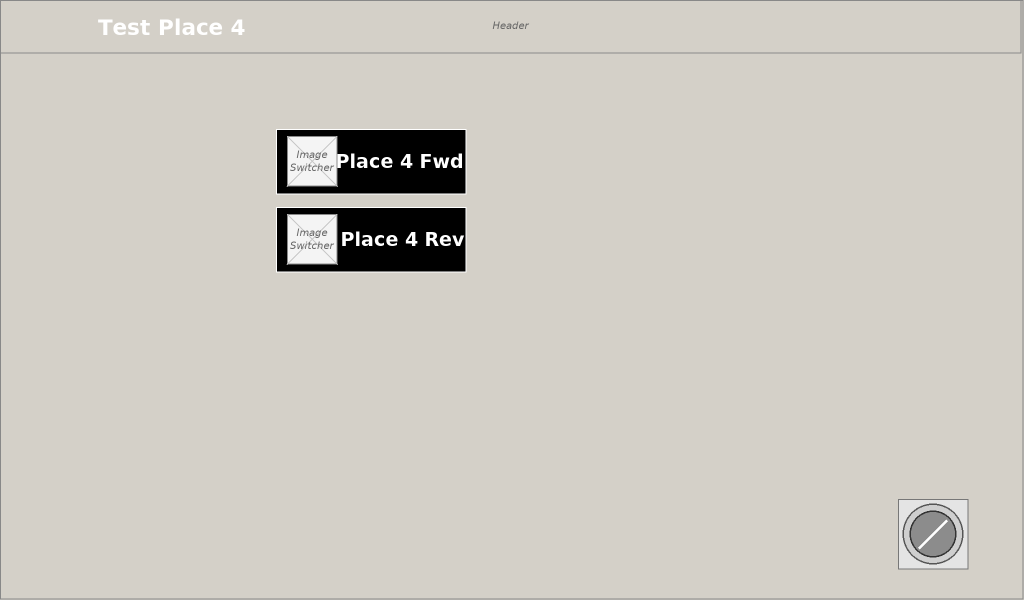
VISUALIZATION Test_Place4  // 1024x600
    Frame (0,-2 1021x55)
        shows Header()
    Label (95,15 250x25), "Test Place 4"
    RotarySwitch (898,499 70x70), variable: HMI_GVL.bTestModeEnablePlacing4, behaviour: TOGGLE, style: Switch-RotarySwitch-Gray
    RoundedRectangle (276,129 190x65)
        toggle Status_GVL.stMotor_Placing4.iTestForward
    Label (331,149 137x25), "Place 4 Fwd"
    ImageSwitcher (287,136 50x50), variable: Status_GVL.stMotor_Placing4.iTestForward, behaviour: TOGGLE
    RoundedRectangle (276,207 190x65)
        toggle Status_GVL.stMotor_Placing4.iTestReverse
    Label (334,227 137x25), "Place 4 Rev"
    ImageSwitcher (287,214 50x50), variable: Status_GVL.stMotor_Placing4.iTestReverse, behaviour: TOGGLE
END_VISUALIZATION

(* stored: Version 1.1.0.1, ProductVersion 3.1.4024.12
   Visu Test_Place4: Id {a17f2ac8-974b-4a4b-beaf-d79f2663683f} *)
